FUNCTION FC_ToBoolArray
VAR_INPUT
	RegSource : POINTER TO BYTE;
	RegDest	  : POINTER TO BOOL;
	Size : UINT;
END_VAR
VAR
	i 	: LWORD;
	j 	: DINT;
	reg : BYTE;
END_VAR

FOR i:=0 TO Size-1 DO
	FOR j:= 0 TO 7 DO
		RegDest^ := TO_BOOL(PBYTE_TO_BYTE((RegSource+i)) AND SHL (1,j));	
		RegDest := RegDest+1;
	END_FOR
END_FOR

END_FUNCTION

(* stored: Version 1.1.0.1, ProductVersion 3.1.4024.13
   POU FC_ToBoolArray: Id {0c1fd8a6-e1fc-45b5-a58b-944b0db3d23a}, SpecialFunc None *)
